(* Schneider Machine Expert - Basic project exercise_4.1, file version 2.9.0.0 *)
(* ProjectInformations: Name=Novo projeto *)

HARDWARE
  Cpu 0: TM221C24R
  EthernetConfiguration: NetworkName=M221, IpAllocationMode=FixedAddress, IpAddress=0.0.0.0, SubnetMask=0.0.0.0
  SerialLineConfiguration: Baud=Baud19200, Parity=ParityEven, DataBits=DataBits8, StopBits=StopBits1, PhysicalMedium=PhysicalMediumRs485, TransmissionMode=TransmissionModeModbusRtu, SlaveId=1, Addressing=SlaveAddressing
  MastTask: UsePeriodScanMode=false, PeriodScan=100
  FastTask: Period=255
  CpuBehavior: StartingMode=StartAsPreviousState, AutoSaveRamOnEeprom=true, WatchdogPeriod=250

SYMBOLS  (address, symbol, comment, settings)
  %M0       SIG_E1_E2
  %M1       SIG_E2_E3
  %M2       SIG_E3_E4
  %M3       SIG_E4_E1
  %M11      SIG_OUT_SEM_HOR_VERD
  %M12      SIG_OUT_SEM_HOR_AMA
  %M13      SIG_OUT_SEM_HOR_VERM
  %M15      SIG_OUT_SEM_VERT_VERD
  %M16      SIG_OUT_SEM_VERT_AMA
  %M17      SIG_OUT_SEM_VERT_VERM
  %X1       E1
  %X2       E2
  %X3       E3
  %X4       E4
  %TM0      FT_E1_E2  [Preset=10, Base=OneSecond]
  %TM1      FT_E2_E3  [Preset=3, Base=OneSecond]
  %TM2      FT_E3_E4  [Preset=10, Base=OneSecond]
  %TM3      FT_E4_E1  [Preset=3, Base=OneSecond]
  %Q0.1     OUT_SEM_HOR_VERD
  %Q0.2     OUT_SEM_HOR_AMA
  %Q0.3     OUT_SEM_HOR_VERM
  %Q0.5     OUT_SEM_VERT_VERD
  %Q0.6     OUT_SEM_VERT_AMA
  %Q0.7     OUT_SEM_VERT_VERM

GRAFCET Grafcet POU
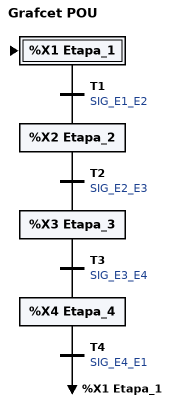
  INITIAL_STEP %X1  (* Etapa_1 *)
  STEP %X2  (* Etapa_2 *)
  STEP %X3  (* Etapa_3 *)
  STEP %X4  (* Etapa_4 *)
  TRANSITION T1 FROM %X1 TO %X2 := SIG_E1_E2;
  TRANSITION T2 FROM %X2 TO %X3 := SIG_E2_E3;
  TRANSITION T3 FROM %X3 TO %X4 := SIG_E3_E4;
  TRANSITION T4 FROM %X4 TO %X1 := SIG_E4_E1;

TRANSITION T1 (%X1 -> %X2) 
  (* SectionNumber=0 *)

// Rung 0: E1_E2
  LD %M0                  (* SIG_E1_E2 *)
  ENDT
  // as ST:
  //   TRANSITION := SIG_E1_E2;

TRANSITION T2 (%X2 -> %X3) 
  (* SectionNumber=0 *)

// Rung 1: E2_E3
  LD %M1                  (* SIG_E2_E3 *)
  ENDT
  // as ST:
  //   TRANSITION := SIG_E2_E3;

TRANSITION T3 (%X3 -> %X4) 
  (* SectionNumber=0 *)

// Rung 2: E3_E4
  LD %M2                  (* SIG_E3_E4 *)
  ENDT
  // as ST:
  //   TRANSITION := SIG_E3_E4;

TRANSITION T4 (%X4 -> %X1) 
  (* SectionNumber=0 *)

// Rung 3: E4_E1
  LD %M3                  (* SIG_E4_E1 *)
  ENDT
  // as ST:
  //   TRANSITION := SIG_E4_E1;

POU Novo POU
  (* SectionNumber=6 *)

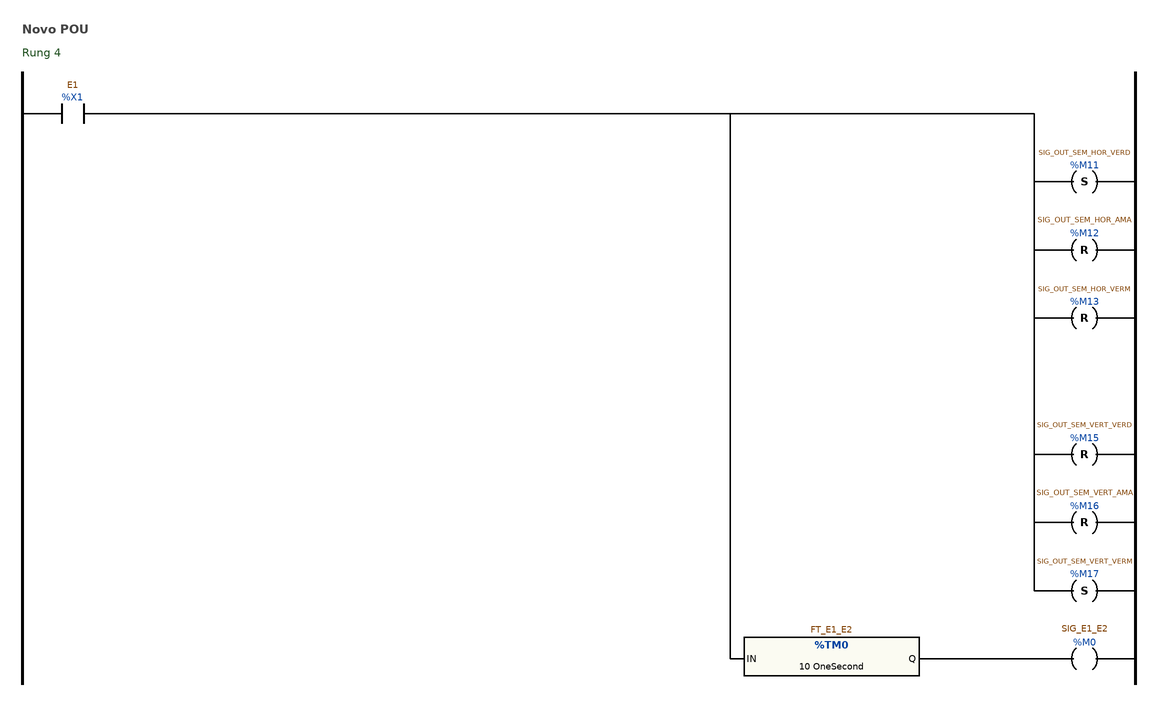

// Rung 4
  LD 1
  MULTIFB
  LD 1
  AND %X1                 (* E1 *)
  ST %MW2009:X0
  LD %MW2009:X0
  S %M11                  (* SIG_OUT_SEM_HOR_VERD *)
  R %M12                  (* SIG_OUT_SEM_HOR_AMA *)
  R %M13                  (* SIG_OUT_SEM_HOR_VERM *)
  R %M15                  (* SIG_OUT_SEM_VERT_VERD *)
  R %M16                  (* SIG_OUT_SEM_VERT_AMA *)
  S %M17                  (* SIG_OUT_SEM_VERT_VERM *)
  BLK %TM0                (* FT_E1_E2 *)
  LD %MW2009:X0
  IN
  OUT_BLK
  LD Q
  ST %M0                  (* SIG_E1_E2 *)
  END_BLK
  MULTIFB
  // as ST:
  //   IF E1 THEN SIG_OUT_SEM_HOR_VERD := TRUE; END_IF;
  //   IF E1 THEN SIG_OUT_SEM_HOR_AMA := FALSE; END_IF;
  //   IF E1 THEN SIG_OUT_SEM_HOR_VERM := FALSE; END_IF;
  //   IF E1 THEN SIG_OUT_SEM_VERT_VERD := FALSE; END_IF;
  //   IF E1 THEN SIG_OUT_SEM_VERT_AMA := FALSE; END_IF;
  //   IF E1 THEN SIG_OUT_SEM_VERT_VERM := TRUE; END_IF;
  //   FT_E1_E2(IN := E1);
  //   SIG_E1_E2 := FT_E1_E2.Q;

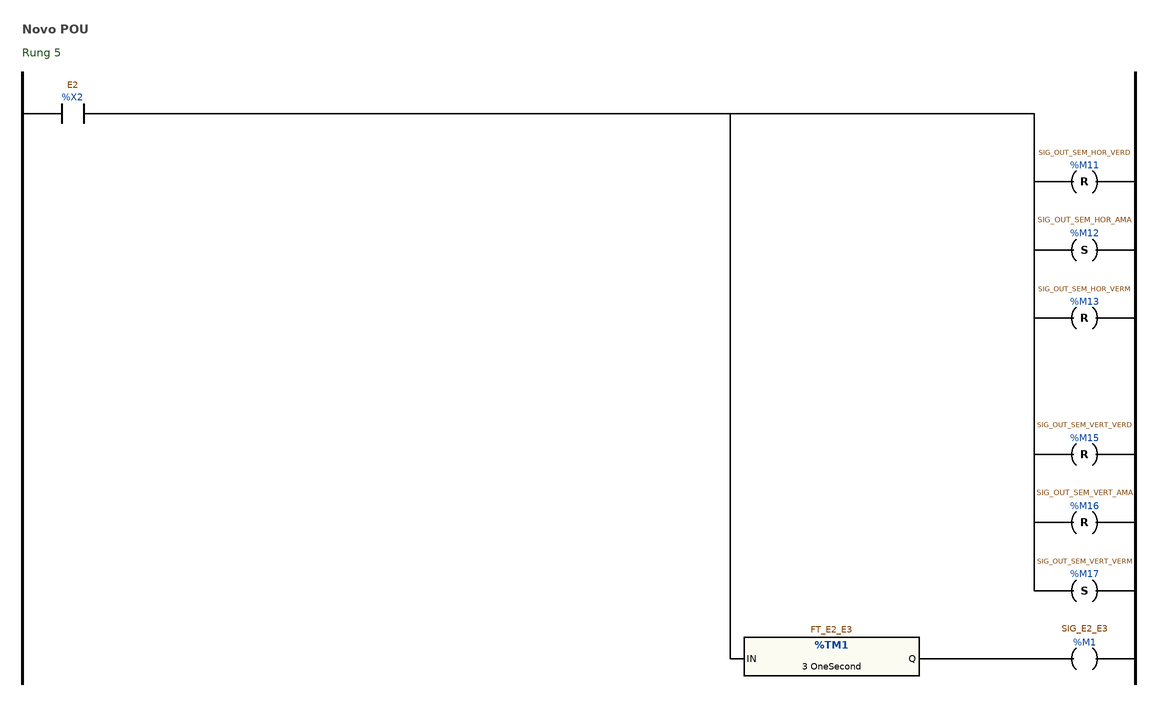

// Rung 5
  LD 1
  MULTIFB
  LD 1
  AND %X2                 (* E2 *)
  ST %MW2009:X0
  LD %MW2009:X0
  R %M11                  (* SIG_OUT_SEM_HOR_VERD *)
  S %M12                  (* SIG_OUT_SEM_HOR_AMA *)
  R %M13                  (* SIG_OUT_SEM_HOR_VERM *)
  R %M15                  (* SIG_OUT_SEM_VERT_VERD *)
  R %M16                  (* SIG_OUT_SEM_VERT_AMA *)
  S %M17                  (* SIG_OUT_SEM_VERT_VERM *)
  BLK %TM1                (* FT_E2_E3 *)
  LD %MW2009:X0
  IN
  OUT_BLK
  LD Q
  ST %M1                  (* SIG_E2_E3 *)
  END_BLK
  MULTIFB
  // as ST:
  //   IF E2 THEN SIG_OUT_SEM_HOR_VERD := FALSE; END_IF;
  //   IF E2 THEN SIG_OUT_SEM_HOR_AMA := TRUE; END_IF;
  //   IF E2 THEN SIG_OUT_SEM_HOR_VERM := FALSE; END_IF;
  //   IF E2 THEN SIG_OUT_SEM_VERT_VERD := FALSE; END_IF;
  //   IF E2 THEN SIG_OUT_SEM_VERT_AMA := FALSE; END_IF;
  //   IF E2 THEN SIG_OUT_SEM_VERT_VERM := TRUE; END_IF;
  //   FT_E2_E3(IN := E2);
  //   SIG_E2_E3 := FT_E2_E3.Q;

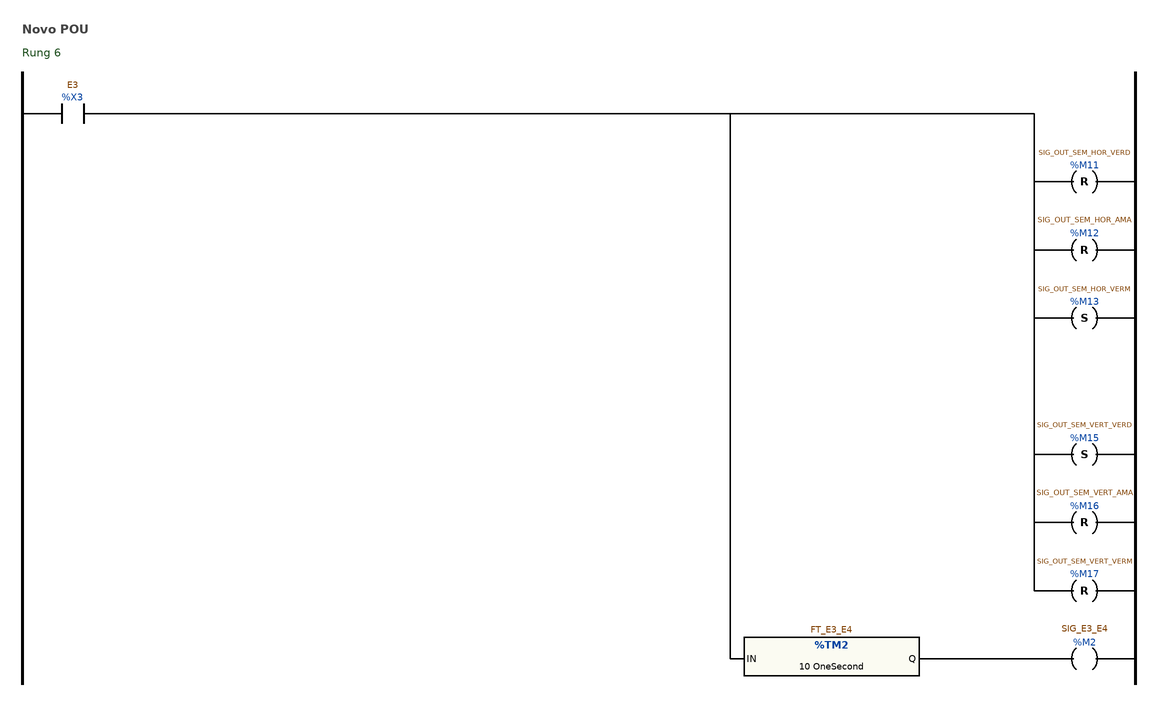

// Rung 6
  LD 1
  MULTIFB
  LD 1
  AND %X3                 (* E3 *)
  ST %MW2009:X0
  LD %MW2009:X0
  R %M11                  (* SIG_OUT_SEM_HOR_VERD *)
  R %M12                  (* SIG_OUT_SEM_HOR_AMA *)
  S %M13                  (* SIG_OUT_SEM_HOR_VERM *)
  S %M15                  (* SIG_OUT_SEM_VERT_VERD *)
  R %M16                  (* SIG_OUT_SEM_VERT_AMA *)
  R %M17                  (* SIG_OUT_SEM_VERT_VERM *)
  BLK %TM2                (* FT_E3_E4 *)
  LD %MW2009:X0
  IN
  OUT_BLK
  LD Q
  ST %M2                  (* SIG_E3_E4 *)
  END_BLK
  MULTIFB
  // as ST:
  //   IF E3 THEN SIG_OUT_SEM_HOR_VERD := FALSE; END_IF;
  //   IF E3 THEN SIG_OUT_SEM_HOR_AMA := FALSE; END_IF;
  //   IF E3 THEN SIG_OUT_SEM_HOR_VERM := TRUE; END_IF;
  //   IF E3 THEN SIG_OUT_SEM_VERT_VERD := TRUE; END_IF;
  //   IF E3 THEN SIG_OUT_SEM_VERT_AMA := FALSE; END_IF;
  //   IF E3 THEN SIG_OUT_SEM_VERT_VERM := FALSE; END_IF;
  //   FT_E3_E4(IN := E3);
  //   SIG_E3_E4 := FT_E3_E4.Q;

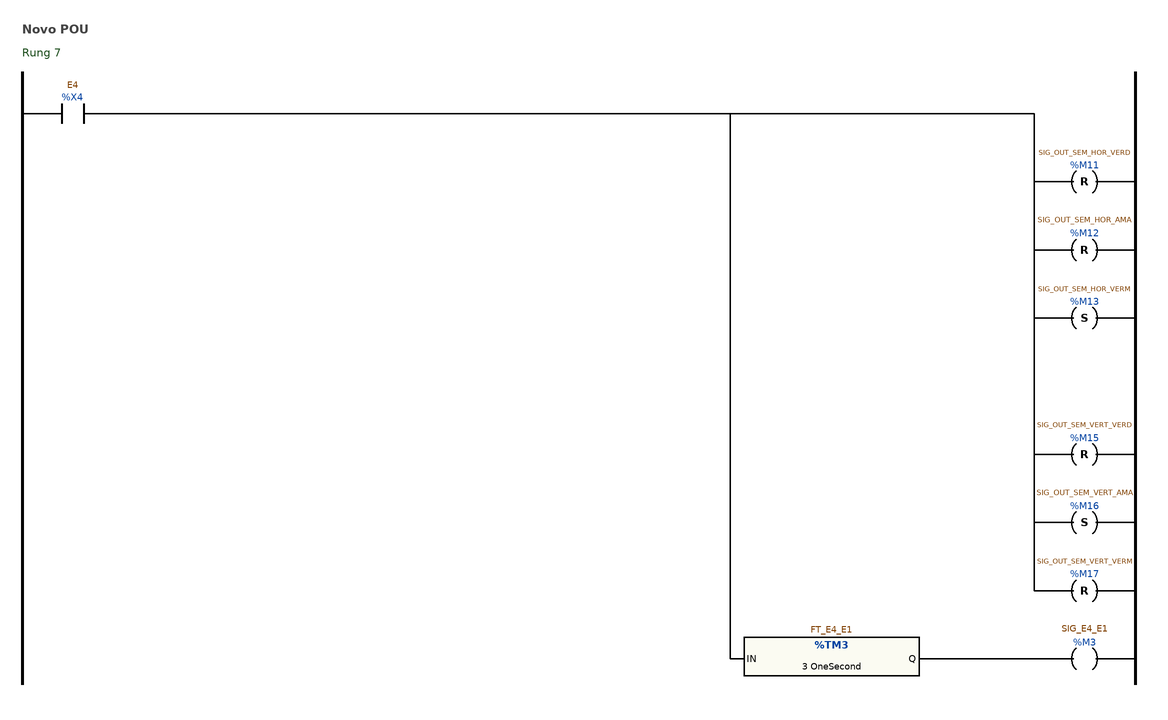

// Rung 7
  LD 1
  MULTIFB
  LD 1
  AND %X4                 (* E4 *)
  ST %MW2009:X0
  LD %MW2009:X0
  R %M11                  (* SIG_OUT_SEM_HOR_VERD *)
  R %M12                  (* SIG_OUT_SEM_HOR_AMA *)
  S %M13                  (* SIG_OUT_SEM_HOR_VERM *)
  R %M15                  (* SIG_OUT_SEM_VERT_VERD *)
  S %M16                  (* SIG_OUT_SEM_VERT_AMA *)
  R %M17                  (* SIG_OUT_SEM_VERT_VERM *)
  BLK %TM3                (* FT_E4_E1 *)
  LD %MW2009:X0
  IN
  OUT_BLK
  LD Q
  ST %M3                  (* SIG_E4_E1 *)
  END_BLK
  MULTIFB
  // as ST:
  //   IF E4 THEN SIG_OUT_SEM_HOR_VERD := FALSE; END_IF;
  //   IF E4 THEN SIG_OUT_SEM_HOR_AMA := FALSE; END_IF;
  //   IF E4 THEN SIG_OUT_SEM_HOR_VERM := TRUE; END_IF;
  //   IF E4 THEN SIG_OUT_SEM_VERT_VERD := FALSE; END_IF;
  //   IF E4 THEN SIG_OUT_SEM_VERT_AMA := TRUE; END_IF;
  //   IF E4 THEN SIG_OUT_SEM_VERT_VERM := FALSE; END_IF;
  //   FT_E4_E1(IN := E4);
  //   SIG_E4_E1 := FT_E4_E1.Q;

POU Saídas
  (* SectionNumber=7 *)

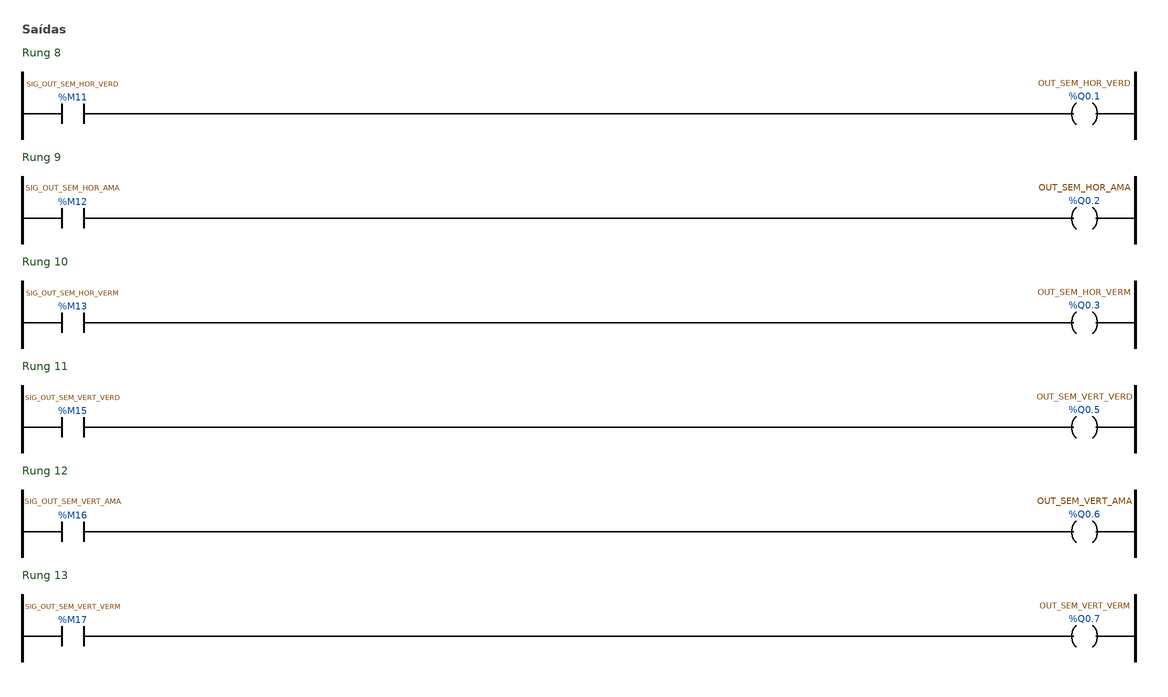

// Rung 8
  LD %M11                 (* SIG_OUT_SEM_HOR_VERD *)
  ST %Q0.1                (* OUT_SEM_HOR_VERD *)
  // as ST:
  //   OUT_SEM_HOR_VERD := SIG_OUT_SEM_HOR_VERD;

// Rung 9
  LD %M12                 (* SIG_OUT_SEM_HOR_AMA *)
  ST %Q0.2                (* OUT_SEM_HOR_AMA *)
  // as ST:
  //   OUT_SEM_HOR_AMA := SIG_OUT_SEM_HOR_AMA;

// Rung 10
  LD %M13                 (* SIG_OUT_SEM_HOR_VERM *)
  ST %Q0.3                (* OUT_SEM_HOR_VERM *)
  // as ST:
  //   OUT_SEM_HOR_VERM := SIG_OUT_SEM_HOR_VERM;

// Rung 11
  LD %M15                 (* SIG_OUT_SEM_VERT_VERD *)
  ST %Q0.5                (* OUT_SEM_VERT_VERD *)
  // as ST:
  //   OUT_SEM_VERT_VERD := SIG_OUT_SEM_VERT_VERD;

// Rung 12
  LD %M16                 (* SIG_OUT_SEM_VERT_AMA *)
  ST %Q0.6                (* OUT_SEM_VERT_AMA *)
  // as ST:
  //   OUT_SEM_VERT_AMA := SIG_OUT_SEM_VERT_AMA;

// Rung 13
  LD %M17                 (* SIG_OUT_SEM_VERT_VERM *)
  ST %Q0.7                (* OUT_SEM_VERT_VERM *)
  // as ST:
  //   OUT_SEM_VERT_VERM := SIG_OUT_SEM_VERT_VERM;
